INTERFACE iCounter

METHOD PUBLIC CmdResetValue : BOOL
END_METHOD

METHOD PUBLIC CmdSetValue : BOOL
VAR_INPUT
	Value : UDINT ;
END_VAR
END_METHOD

PROPERTY PUBLIC CountValue : UDINT
GET
END_GET
END_PROPERTY

END_INTERFACE

(* stored: Version 1.1.0.1, ProductVersion 3.1.4024.10
   Itf iCounter: Id {99eb9e42-0844-0373-3007-aa469c33325f}
   Method CmdResetValue: Id {c8f65e43-e9db-0d46-368c-11e932d8e453}
   Method CmdSetValue: Id {a14f7d20-1980-0f0b-0f0b-f99755f732db}
   Property CountValue: Id {46a841e9-a25b-0322-3b9f-ecdddc9a6e82}
   Get Get: Id {cee3cabc-7739-0dbc-1e49-aaf81b0685a8} *)
